FUNCTION PlainFunction : BOOL
VAR_INPUT
END_VAR
VAR
END_VAR

END_FUNCTION

(* stored: Version 1.1.0.1, ProductVersion 3.1.4024.11
   POU PlainFunction: Id {245635d0-7d54-4aa8-92df-875383b63265}, SpecialFunc None *)
